PROGRAM valve_control
VAR
	//Repeat for each valve?
	pump_1_enable: BOOL;
	pump_1_auto_request: BOOL;
	pump_1_cip_request: BOOL;
	pump_1_manual_request: BOOL;
	pump_1_stop_request: BOOL;
	pump_1_intlk: BOOL;
	gen_alm_active: BOOL;
	ed_routine_auto: BOOL;
	ed_routine_cip: BOOL;
	ed_routine_manual: BOOL;
	valve_1_auto_request: BOOL;
	valve_1_cip_request: BOOL;
	valve_1_manual_request: BOOL;
	valve_1_intlk: BOOL;
	valve_1_stop_request: BOOL;
	valve_1_enable: BOOL;
END_VAR

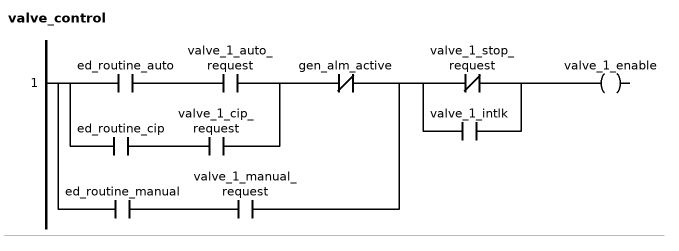
// NETWORK 1
valve_1_enable := ((ed_routine_auto AND valve_1_auto_request OR ed_routine_cip AND valve_1_cip_request) AND NOT gen_alm_active OR ed_routine_manual AND valve_1_manual_request) AND (NOT valve_1_stop_request OR valve_1_intlk);

END_PROGRAM

(* stored: Version 1.1.0.1, ProductVersion 3.1.4024.12
   POU valve_control: Id {359c8254-c75f-419b-be16-97d4ba9197db}, SpecialFunc None *)
